VAR_GLOBAL
	G_xAutoMode:					BOOL;
	G_nOperationMode:				INT:=1;
	
	G_nSequenceLength:				INT;
	G_xSequenceRowReady:			BOOL;
	G_xSequenceRowDone:				BOOL;
	
	G_xManualMoveMode:				BOOL:=TRUE;											//1:= continous, 0:= stepper
	G_lrOverride:					LREAL;												//Main overrride value
	G_lrManualOverride:				LREAL:=20;
	G_lrStepSize:					LREAL:=0.1;
	G_lrMaximumVelocity:			LREAL:=600;
	
	G_sActualPosition:				tsCoordinate;										//Actual coordinate
	G_sTargetPosition:				tsCoordinate;										//Actual target position
	
	G_sAxisReady:					tsCoordinateBool;									//Axis ready to move state container
	G_sAxisDone:					tsCoordinateBool;									//Axis done state container
	G_sAckAxisDone:					tsCoordinateBool;									//Axis done acknowledge container
	
	G_sAxisJogForward:				tsCoordinateBool;									//Axis jog forward
	G_sAxisJogBackward:				tsCoordinateBool;									//Axis jog backward
	
	G_sStartToPos:					tsCoordinateBool;									//Start to position
	G_xPowerOn: 					BOOL:=TRUE;
	
	//SFC Variables
	SFCPause:BOOL;
	SFCReset:BOOL;
	
END_VAR

(* stored: Version 1.1.0.1, ProductVersion 3.1.4022.18
   GVL MAIN_GVL: Id {8a90cd30-80b2-4b65-a07c-67fb08b99178} *)
